ABB RAPID module: Wobj_wobj_C.mod

MODULE Wobj_wobj_C
	! Points are read in order of declaration.
  ! Please do not change the order of points!

  LOCAL PERS robtarget pWobj_U_PointX1:=[[-1109.108,-2083.159,-728.8731],[0.000221819529542699,-0.727543115615845,0.686061441898346,0.000849400239530951],[-2,-1,1,0],[0,9E+09,9E+09,9E+09,9E+09,9E+09]];
	LOCAL PERS robtarget pWobj_U_PointX2:=[[-713.5533,-2083.083,-728.8806],[0.000235550745856017,-0.727545440196991,0.686058938503265,0.000853651028592139],[-2,-1,1,0],[0,9E+09,9E+09,9E+09,9E+09,9E+09]];
	LOCAL PERS robtarget pWobj_U_PointY1:=[[-741.7236,-1965.849,-728.8785],[0.000231423880904913,-0.727521300315857,0.686084508895874,0.000853470817673951],[-2,-1,1,0],[0,9E+09,9E+09,9E+09,9E+09,9E+09]];

ENDMODULE
